PROGRAM MAIN
VAR
    Initialize	:	BOOL := TRUE;

    fbLogHandler : FB_LogHandler;
    fbEcatDiag : FB_EcatDiagWrapper;

	idx: UINT;
	
	//System Time
	 {attribute 'pytmc' := '
        pv: @(PREFIX)SystemDT
        io: i
     '}
	SystemTime:DINT;
	fbTime : FB_LocalSystemTime := ( bEnable := TRUE, dwCycle := 1 ); //Get current system time, used for override
	fbTime_to_UTC: FB_TzSpecificLocalTimeToSystemTime;
	fbGetTimeZone: FB_GetTimeZoneInformation;
END_VAR

//Arbiter PLC

IF Initialize THEN
    Initialize := FALSE;
	
	// Setting apertures to zero for now
	FOR idx := 1 TO PMPS_GVL.MAX_APERTURES DO
		PMPS_GVL.stCurrentBeamParameters.astApertures[idx].Height := 0;
		PMPS_GVL.stCurrentBeamParameters.astApertures[idx].Width := 0;
	END_FOR
END_IF

// Ethercat Diagnostics
fbEcatDiag();

CurrentBPUpdate();

///////////////////////////////////////////////////
// This code should be disabled or removed in deployment
// Might have a switch to change to simulation mode
MachineSimulation();
//Testing();
///////////////////////////////////////////////////

// PMPS Functionality

PMPS_Arbiter();
A_SystemTime();

P_SATT();

fbLogHandler();

ACTION A_SystemTime:
//Get local System Time
fbTime(sNetID:='');
//Get Time Zone
fbGetTimeZone(sNetID:='',bExecute:=TRUE,tTimeout:=T#10S);
//change local time to UTC to be compatible with unix time epoch widget
fbTime_to_UTC(in:= fbTime.systemTime , tzInfo:=fbGetTimeZone.tzInfo);

SystemTime:= TO_DINT(TO_DT(SystemTime_TO_DT(fbTime_to_UTC.out)));
END_ACTION

ACTION Initialize:

END_ACTION

END_PROGRAM

(* stored: Version 1.1.0.1, ProductVersion 3.1.4022.18
   POU MAIN: Id {8a7bcfd2-1a2b-4363-aa47-c19391bf1f9c}, SpecialFunc None
   Action A_SystemTime: Id {a361e090-c874-45d8-82ab-48f0371b64c5}
   Action Initialize: Id {b0ee480a-3d4b-001d-04c4-43cdc47895c8} *)
